// TIA Portal V17 export
// export: Created 2024-09-02T12:50:06.2619829Z, ExportSetting WithDefaults, DisplayName Totally Integrated Automation Portal, DisplayVersion V17, DisplayName TIA Portal Openness, DisplayVersion V17, DisplayName TIA Portal Version Control Interface, DisplayVersion V17, DisplayName STEP 7 Professional, DisplayVersion V17, DisplayName STEP 7 Safety, DisplayVersion V17, DisplayName WinCC Professional, DisplayVersion V17
FUNCTION_BLOCK "GraFB9_FG01_Home_OP70"   // FB1289, GRAPH
VERSION : 0.1
// stored: AcknowledgeErrorsRequired true, AutoNumber false, GraphVersion 4.0, InitialValuesAcquisition false, IsIECCheckEnabled false, LanguageInNetworks LAD, LockOperatingMode false, PermanentILProcessingInMANMode true, SetENOAutomatically false, SkipSteps false, UDAEnableTagReadback false, WithAlarmHandling true
   // inherited from GRAPH_BASE
   VAR
      OFF_SQ_BASE : Bool;
   END_VAR
   VAR_INPUT
      OFF_SQ { ExternalWritable := 'False'} : Bool := false;   // Kette ausschalten / Turn sequence off
      INIT_SQ { ExternalWritable := 'False'} : Bool := false;   // Kette in Initialzustand versetzen / Set sequence to initial state
      ACK_EF { ExternalWritable := 'False'} : Bool := false;   // Alle Fehler und Störungen quittieren / Acknowledge all errors and faults
      S_PREV { ExternalWritable := 'False'} : Bool := false;   // Vorherigen Schritt am Parameter S_NO ausgeben / Output previous step in parameter S_NO
      S_NEXT { ExternalWritable := 'False'} : Bool := false;   // Nächsten Schritt am Parameter S_NO anzeigen / Indicate next step in parameter S_NO
      SW_AUTO { ExternalWritable := 'False'} : Bool := false;   // Automtischer Betrieb / Automatic mode
      SW_TAP { ExternalWritable := 'False'} : Bool := false;   // Halbautomatisch/Weiterschalten mit Transition / Semiautomatic/switch with transition
      SW_TOP { ExternalWritable := 'False'} : Bool := false;   // Halbautomatisch/Ignoriere Transition / Semiautomatic/ignore transition
      SW_MAN { ExternalWritable := 'False'} : Bool := false;   // Handbetrieb / Manual mode
      S_SEL { ExternalWritable := 'False'} : Int := 0;   // Schritt auswählen, der an S_NO ausgegeben werden soll / Select step to be output to S_NO
      S_ON { ExternalWritable := 'False'} : Bool := false;   // Schritt aktivieren, der an Parameter S_NO anliegt / Activate step indicated in S_NO
      S_OFF { ExternalWritable := 'False'} : Bool := false;   // Schritt deaktivieren, der an Parameter S_NO anliegt / Deactivate step indicated S_NO
      T_PUSH { ExternalWritable := 'False'} : Bool := false;   // Schaltfreigabe für Transition im halbautomatischen Betrieb / Enable transition to switch in semi automatic mode
   END_VAR
   VAR_OUTPUT
      S_NO { ExternalWritable := 'False'} : Int := 0;   // Schrittnummer / Step number
      S_MORE { ExternalWritable := 'False'} : Bool := false;   // Weitere Schritte sind vorhanden und können in S_NO angezeigt werden. / More steps are available and can be shown in S_NO
      S_ACTIVE { ExternalWritable := 'False'} : Bool := false;   // Schritt, der an Parameter S_NO angezeigt wird, ist aktiv / Step indicated in S_NO is active
      ERR_FLT { ExternalWritable := 'False'} : Bool := false;   // Sammelfehler Interlock oder Supervision / Interlock or supervision group error
      AUTO_ON { ExternalWritable := 'False'} : Bool := false;   // Automatischer Betrieb eingeschaltet / Automatic mode is active
      TAP_ON { ExternalWritable := 'False'} : Bool := false;   // Halbautomatischer Betrieb/Schritt mit Transition eingeschaltet / Semiautomatic mode/step with transition enabled
      TOP_ON { ExternalWritable := 'False'} : Bool := false;   // Halbautomatischer Betrieb/Ignoriere Transition eingeschaltet / Semiautomatic mode/ignore transition enabled
      MAN_ON { ExternalWritable := 'False'} : Bool := false;   // Handbetrieb eingeschaltet / Manual mode is active
   END_VAR
   VAR
      extBlock { S7_SetPoint := 'True'} : "LTLL_ManualGraphExt";
   END_VAR
BEGIN
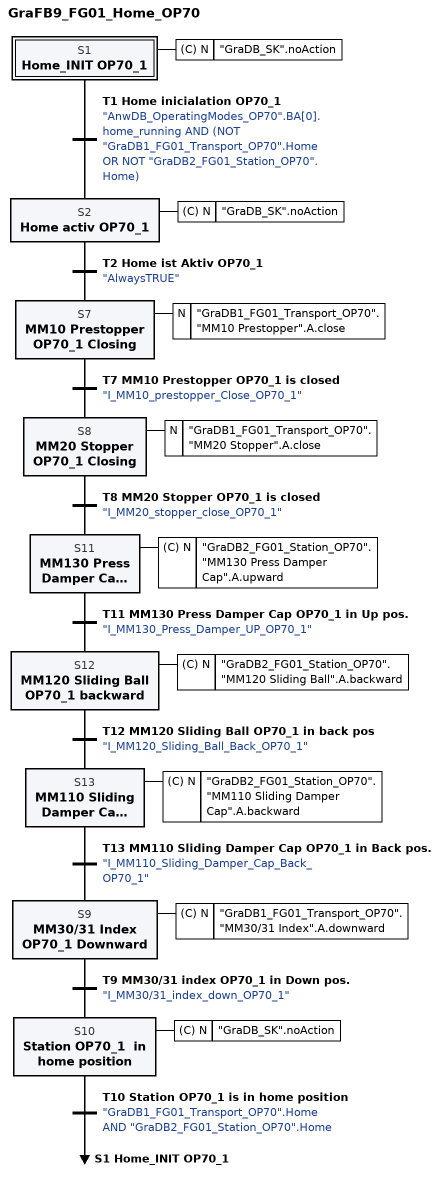
   // permanent pre-instructions
   NETWORK 1
   TITLE = HMI Lite Pass on data / HMI Lite Daten weiterreichen
      #extBlock.input := "LTLL_ManualGraphControl_OP70".screen[0].input;
   NETWORK 2
   TITLE = Instance DB Name query and pass on / Instanz DB Name abfragen und weiterreichen
      GetInstanceName(size := 0, OUT => #extBlock.input.instanceName);
   NETWORK 3
   TITLE = SK Mode
      "SysFC_SQ_Mode"(iFKT := 0, iTmsHalt := false, ioMOP := #RT_DATA.MOP);

   // sequencer 1: basic position drive / Grundstellungsfahrt
   INITIAL_STEP "Home_INIT OP70_1":   // S1, max time T#10S, warning time T#7S: Step commentary / Schrittkommentar
      interlock C := (none);   // Initialschritt / initial step
      supervision V := (none);   // Initialschritt / initial step
      (C)     N    "GraDB_SK".noAction
   END_STEP
   TRANSITION "Home inicialation OP70_1" FROM "Home_INIT OP70_1" TO "Home activ OP70_1"   // T1
      := "AnwDB_OperatingModes_OP70".BA[0].home_running AND (NOT "GraDB1_FG01_Transport_OP70".Home OR NOT "GraDB2_FG01_Station_OP70".Home);
   END_TRANSITION
   STEP "Station OP70_1  in home position":   // S10, max time T#10S, warning time T#7S
      supervision V := NOT #"Station OP70_1 is in home position".TT AND (#"Station OP70_1  in home position".U > T#5S);
      (C)     N    "GraDB_SK".noAction
   END_STEP
   TRANSITION "Station OP70_1 is in home position" FROM "Station OP70_1  in home position" TO "Home_INIT OP70_1"   // T10, jump
      := "GraDB1_FG01_Transport_OP70".Home AND "GraDB2_FG01_Station_OP70".Home;
   END_TRANSITION
   STEP "Home activ OP70_1":   // S2, max time T#10S, warning time T#7S
      supervision V := NOT #"Home ist Aktiv OP70_1".TT AND (#"Home activ OP70_1".U > T#5S);
      (C)     N    "GraDB_SK".noAction
   END_STEP
   TRANSITION "Home ist Aktiv OP70_1" FROM "Home activ OP70_1" TO "MM10 Prestopper OP70_1 Closing"   // T2
      := "AlwaysTRUE";
   END_TRANSITION
   STEP "MM10 Prestopper OP70_1 Closing":   // S7, max time T#10S, warning time T#7S
      supervision V := NOT #"MM10 Prestopper OP70_1 is closed".TT AND (#"MM10 Prestopper OP70_1 Closing".U > T#5S);
              N    "GraDB1_FG01_Transport_OP70"."MM10 Prestopper".A.close
   END_STEP
   TRANSITION "MM10 Prestopper OP70_1 is closed" FROM "MM10 Prestopper OP70_1 Closing" TO "MM20 Stopper OP70_1 Closing"   // T7
      := "I_MM10_prestopper_Close_OP70_1";
   END_TRANSITION
   STEP "MM20 Stopper OP70_1 Closing":   // S8, max time T#10S, warning time T#7S
      supervision V := NOT #"MM20 Stopper OP70_1 is closed".TT AND (#"MM20 Stopper OP70_1 Closing".U > T#5S);
              N    "GraDB1_FG01_Transport_OP70"."MM20 Stopper".A.close
   END_STEP
   TRANSITION "MM20 Stopper OP70_1 is closed" FROM "MM20 Stopper OP70_1 Closing" TO "MM130 Press Damper Cap OP70_1 Upward"   // T8
      := "I_MM20_stopper_close_OP70_1";
   END_TRANSITION
   STEP "MM30/31 Index OP70_1 Downward":   // S9, max time T#10S, warning time T#7S
      interlock C := "I_MM130_Press_Damper_UP_OP70_1";
      supervision V := NOT #"MM30/31 index OP70_1 in Down pos.".TT AND (#"MM30/31 Index OP70_1 Downward".U > T#5S);
      (C)     N    "GraDB1_FG01_Transport_OP70"."MM30/31 Index".A.downward
   END_STEP
   TRANSITION "MM30/31 index OP70_1 in Down pos." FROM "MM30/31 Index OP70_1 Downward" TO "Station OP70_1  in home position"   // T9
      := "I_MM30/31_index_down_OP70_1";
   END_TRANSITION
   STEP "MM130 Press Damper Cap OP70_1 Upward":   // S11, max time T#10S, warning time T#7S
      interlock C := "AlwaysTRUE";
      supervision V := NOT #"MM130 Press Damper Cap OP70_1 in Up pos.".TT AND (#"MM130 Press Damper Cap OP70_1 Upward".U > T#5S);
      (C)     N    "GraDB2_FG01_Station_OP70"."MM130 Press Damper Cap".A.upward
   END_STEP
   TRANSITION "MM130 Press Damper Cap OP70_1 in Up pos." FROM "MM130 Press Damper Cap OP70_1 Upward" TO "MM120 Sliding Ball OP70_1 backward"   // T11
      := "I_MM130_Press_Damper_UP_OP70_1";
   END_TRANSITION
   STEP "MM120 Sliding Ball OP70_1 backward":   // S12, max time T#10S, warning time T#7S
      interlock C := "AlwaysTRUE";
      supervision V := NOT #"MM120 Sliding Ball OP70_1 in back pos".TT AND (#"MM120 Sliding Ball OP70_1 backward".U > T#5S);
      (C)     N    "GraDB2_FG01_Station_OP70"."MM120 Sliding Ball".A.backward
   END_STEP
   TRANSITION "MM120 Sliding Ball OP70_1 in back pos" FROM "MM120 Sliding Ball OP70_1 backward" TO "MM110 Sliding Damper Cap OP70_1 Backward"   // T12
      := "I_MM120_Sliding_Ball_Back_OP70_1";
   END_TRANSITION
   STEP "MM110 Sliding Damper Cap OP70_1 Backward":   // S13, max time T#10S, warning time T#7S
      interlock C := "I_MM130_Press_Damper_UP_OP70_1";
      supervision V := NOT #"MM110 Sliding Damper Cap OP70_1 in Back pos.".TT AND (#"MM110 Sliding Damper Cap OP70_1 Backward".U > T#5S);
      (C)     N    "GraDB2_FG01_Station_OP70"."MM110 Sliding Damper Cap".A.backward
   END_STEP
   TRANSITION "MM110 Sliding Damper Cap OP70_1 in Back pos." FROM "MM110 Sliding Damper Cap OP70_1 Backward" TO "MM30/31 Index OP70_1 Downward"   // T13
      := "I_MM110_Sliding_Damper_Cap_Back_OP70_1";
   END_TRANSITION

   // permanent post-instructions
   NETWORK 1
   TITLE = Move interlocks from Ext block to ManualGraphControl DB / Interlocks vom Ext-Block zum ManualGraphControl DB rangieren
      "LTLL_ManualGraphInterlock"(ManualGraphExtOutput := #extBlock.output,
                              ManualGraphControlScreen := "LTLL_ManualGraphControl_OP70".screen[0]);
   NETWORK 2
   TITLE = Report step error / Schrittkettenfehler melden
      "SysFC_NumOfSQErrors"(FLT := #RT_DATA.SQ_FLAGS.ERR_FLT,
                            Fault_SQ := "AnwDB_OperatingModes_OP70".BA[0].error_report_SK,
                            NumOf_Fault_SQ := "AnwDB_ZP_Alarm_OP70".FaultsNoSK_ST1);
   NETWORK 3
   TITLE = SK in home position / SK in Grundstellung
      "GraDB_Home".OP70_1.Home_SK := #"Home_INIT OP70_1".X;
END_FUNCTION_BLOCK
